# EPICS substitutions: iocBoot/ioc-xrt-xcsimb3/ioc-xrt-xcsimb3.substitutions
# IOC archive file
## Replace TST:R40:IOC:22 with the PV prefix used for
## iocAdmin PV's on this IOC

# Generate IOC archive request
file archive_ipimbIoc.archive
{
	{ IOC = "XRT:R38:IOC:43" }
}
